Fanuc KAREL source: kt00901.KL

-- PROVISIONAL review KL for V770-1; original PC SHA256 59079c55b3b4a182dd78534cf9caa10bba829ffb9b68672e2a05d65a22f912ce
-- Incomplete behavior may be omitted. Consult companion uncertainty JSON. Do not deploy.
PROGRAM KT00901
%NOLOCKGROUP
VAR
  OUT : BOOLEAN
-- UNRESOLVED_DECL P1 type=000199
-- UNRESOLVED_DECL P2 type=000199
BEGIN
  -- UNRESOLVED_PC offsets 5-28; opcodes 27,22,1C,27,9D,76,23
  -- UNRESOLVED_PC offsets 33-37; opcodes 7F
END KT00901
